(* IEC 61131-3 sources: verifaps-lib/iec-modularization/src/test/resources, 5 files *)

(* ---- program.st ---- *)
FUNCTION_BLOCK FB
VAR_INPUT
	x : INT;
END_VAR
VAR_OUTPUT
	y : INT;
END_VAR
	y := x+6;
END_FUNCTION_BLOCK

PROGRAM PGRM
VAR_INPUT
	x : INT;
END_VAR
VAR_OUTPUT
	y : INT;
END_VAR
VAR
	INST_FB : FB;
END_VAR
	INST_FB.x := 4;
	INST_FB();
	INST_FB.x := INST_FB.y + 2;
	INST_FB();
	y := INST_FB.y;
	IF x > 5 THEN
		y := 6;
	ELSEIF x > 3 THEN
		y := 7;
	ELSE
		y := x;
	END_IF
	y := y + 4;
END_PROGRAM

(* ---- program1.st ---- *)
TYPE
	TestEnum: (First, Second);
END_TYPE

FUNCTION_BLOCK BLOCK_A
	VAR_INPUT  x : INT; END_VAR
	VAR_OUTPUT y : INT; END_VAR
	y := x - INT#4;
END_FUNCTION_BLOCK

FUNCTION_BLOCK BLOCK_B
	VAR_INPUT  x : INT; END_VAR
	VAR_OUTPUT y : INT; END_VAR
	y := x + INT#6;
END_FUNCTION_BLOCK

FUNCTION_BLOCK TON
END_FUNCTION_BLOCK

PROGRAM PGRM
	VAR_INPUT  x      : INT;     END_VAR
	VAR_OUTPUT y      : INT;     END_VAR
	VAR        INST_A : BLOCK_A; END_VAR
	VAR        INST_B : BLOCK_B; END_VAR
	VAR        state  : TestEnum; END_VAR
	VAR  TestTimer : TON; END_VAR

	CASE state OF
		TestEnum#First:
			INST_A.x := INT#4;
		TestEnum#Second:
			INST_A.x := INT#8;
	END_CASE
	TestTimer();
	INST_A.x := x + INT#7;
	IF x > 5 THEN
		INST_A();
	END_IF

	INST_B.x := INST_A.y + INT#9;
	INST_B();

	y := INST_B.y;
END_PROGRAM

(* ---- program2.st ---- *)
FUNCTION_BLOCK BLOCK_A
	VAR_INPUT  x : INT; END_VAR
	VAR_OUTPUT y : INT; END_VAR
	y := x - INT#4;
END_FUNCTION_BLOCK

FUNCTION_BLOCK BLOCK_B
	VAR_INPUT  x : INT; END_VAR
	VAR_OUTPUT y : INT; END_VAR
	y := x + INT#3;
END_FUNCTION_BLOCK

PROGRAM PGRM
	VAR_INPUT  x      : INT;     END_VAR
	VAR_OUTPUT y      : INT;     END_VAR
	VAR        INST_A : BLOCK_A; END_VAR
	VAR        INST_B : BLOCK_B; END_VAR

	INST_A.x := x + INT#7;
	INST_A();

	INST_B.x := INST_A.y + INT#9;
	INST_B();

	y := INST_B.y + INT#3;
END_PROGRAM

(* ---- scenario0.st ---- *)
TYPE
    Magazin_states_t : (Green_Lamp , Init , Interstep , Magazin_Init , Magazin_Init_2 , Slider_Move_Back , Start_Magazin , Step0 , Step1 , convey);
    Crane_states_t : (Crane_Init , Crane_Init_2 , Crane_Lift_Conveyor , Crane_Lift_Magazine , Crane_On_Conveyor , Crane_Stop , Crane_Turn_Left , Init , Interstep , Interstep_2 , Interstep_Check_Workpiece , Magazin_Stop , Start_Crane , TimeDelay , Turn_Right , release);
END_TYPE

FUNCTION_BLOCK Magazin
    VAR_INPUT  CraneDown : BOOL; END_VAR
    VAR_INPUT  CraneOnConveyor : BOOL; END_VAR
    VAR_INPUT  CraneOnMagazin : BOOL; END_VAR
    VAR_INPUT  CraneSucked : BOOL; END_VAR
    VAR_INPUT  CraneUp : BOOL; END_VAR
    VAR_OUTPUT  MagazinGreenLamp : BOOL; END_VAR
    VAR_OUTPUT  MagazinSlider : BOOL; END_VAR
    VAR  SFCInit : BOOL; END_VAR
    VAR_INPUT  SFCReset : BOOL; END_VAR
    VAR_INPUT  SliderMovedOut : BOOL; END_VAR
    VAR_INPUT  SliderNotMovedOut : BOOL; END_VAR
    VAR_INPUT  StartButtonMagazin : BOOL; END_VAR
    VAR_OUTPUT  StartCommandMagazin : BOOL; END_VAR
    VAR_INPUT  StartVar : BOOL; END_VAR
    VAR_INPUT  WorkpieceReady : BOOL; END_VAR
    VAR  _state : Magazin_states_t; END_VAR
    VAR  _transit : BOOL; END_VAR
    VAR  interconnectMagazineStartCommand : BOOL; END_VAR

    CASE _state OF
        Magazin_states_t#Green_Lamp:
            _transit := FALSE;
            MagazinGreenLamp := TRUE;
            interconnectMagazineStartCommand := FALSE;
            IF TRUE THEN
                _transit := TRUE;
                _state := Magazin_states_t#Magazin_Init;
            END_IF;

        Magazin_states_t#Init:
            _transit := FALSE;
            IF TRUE THEN
                _transit := TRUE;
                _state := Magazin_states_t#Start_Magazin;
            END_IF;

        Magazin_states_t#Interstep:
            _transit := FALSE;
            StartCommandMagazin := TRUE;
            IF StartVar THEN
                _transit := TRUE;
                _state := Magazin_states_t#convey;
            END_IF;

        Magazin_states_t#Magazin_Init:
            _transit := FALSE;
            MagazinSlider := TRUE;
            IF TRUE THEN
                _transit := TRUE;
                _state := Magazin_states_t#Magazin_Init_2;
            END_IF;

        Magazin_states_t#Magazin_Init_2:
            _transit := FALSE;
            MagazinSlider := FALSE;
            IF TRUE THEN
                _transit := TRUE;
                _state := Magazin_states_t#Interstep;
            END_IF;

        Magazin_states_t#Slider_Move_Back:
            _transit := FALSE;
            IF ((SliderMovedOut = TRUE) AND (SliderNotMovedOut = FALSE)) THEN
                MagazinSlider := FALSE;
            END_IF;
            IF CraneUp THEN
                _transit := TRUE;
                _state := Magazin_states_t#Step1;
            END_IF;

        Magazin_states_t#Start_Magazin:
            _transit := FALSE;
            MagazinSlider := FALSE;
            MagazinGreenLamp := FALSE;
            StartVar := FALSE;
            StartCommandMagazin := FALSE;
            IF (StartButtonMagazin = TRUE) THEN
                interconnectMagazineStartCommand := TRUE;
            END_IF;
            IF interconnectMagazineStartCommand THEN
                _transit := TRUE;
                _state := Magazin_states_t#Green_Lamp;
            END_IF;

        Magazin_states_t#Step0:
            _transit := FALSE;
            IF CraneDown THEN
                _transit := TRUE;
                _state := Magazin_states_t#Slider_Move_Back;
            END_IF;

        Magazin_states_t#Step1:
            _transit := FALSE;
            IF CraneOnConveyor THEN
                _transit := TRUE;
                _state := Magazin_states_t#Interstep;
            END_IF;

        Magazin_states_t#convey:
            _transit := FALSE;
            IF SliderNotMovedOut THEN
                MagazinSlider := TRUE;
            END_IF;
            IF CraneOnMagazin THEN
                _transit := TRUE;
                _state := Magazin_states_t#Step0;
            END_IF;

            END_CASE
END_FUNCTION_BLOCK

FUNCTION_BLOCK Crane
    VAR_INPUT  CraneDown : BOOL; END_VAR
    VAR_OUTPUT  CraneLower : BOOL; END_VAR
    VAR_INPUT  CraneOnConveyor : BOOL; END_VAR
    VAR_INPUT  CraneOnMagazin : BOOL; END_VAR
    VAR_INPUT  CraneSucked : BOOL; END_VAR
    VAR_OUTPUT  CraneTurnClockwise : BOOL; END_VAR
    VAR_OUTPUT  CraneTurnCounterclockwise : BOOL; END_VAR
    VAR_INPUT  CraneUp : BOOL; END_VAR
    VAR_OUTPUT  MagazinVacuumOff : BOOL; END_VAR
    VAR_OUTPUT  MagazinVacuumOn : BOOL; END_VAR
    VAR  SFCInit : BOOL; END_VAR
    VAR_INPUT  SFCReset : BOOL; END_VAR
    VAR_INPUT  SliderMovedOut : BOOL; END_VAR
    VAR_INPUT  SliderNotMovedOut : BOOL; END_VAR
    VAR_INPUT  StartButtonMagazin : BOOL; END_VAR
    VAR_OUTPUT  StartCommandCrane : BOOL; END_VAR
    VAR_INPUT  StartVar : BOOL; END_VAR
    VAR  TimeDelay_Timer : TON; END_VAR
    VAR  TimeDelay_Timer_Duration : INT := INT#50; END_VAR
    VAR  TimeDelay_Timer_interconnect : BOOL; END_VAR
    VAR_INPUT  WorkpieceReady : BOOL; END_VAR
    VAR  _state : Crane_states_t; END_VAR
    VAR  _transit : BOOL; END_VAR
    VAR  interconnectCraneStartCommand : BOOL; END_VAR

    CASE _state OF
        Crane_states_t#Crane_Init:
            _transit := FALSE;
            CraneLower := TRUE;
            interconnectCraneStartCommand := FALSE;
            IF CraneDown THEN
                _transit := TRUE;
                _state := Crane_states_t#Crane_Init_2;
            END_IF;

        Crane_states_t#Crane_Init_2:
            _transit := FALSE;
            CraneLower := FALSE;
            IF CraneUp THEN
                _transit := TRUE;
                _state := Crane_states_t#Interstep;
            END_IF;

        Crane_states_t#Crane_Lift_Conveyor:
            _transit := FALSE;
            CraneLower := FALSE;
            IF TRUE THEN
                _transit := TRUE;
                _state := Crane_states_t#Interstep;
            END_IF;

        Crane_states_t#Crane_Lift_Magazine:
            _transit := FALSE;
            CraneLower := FALSE;
            IF CraneUp THEN
                _transit := TRUE;
                _state := Crane_states_t#Crane_Turn_Left;
            END_IF;

        Crane_states_t#Crane_On_Conveyor:
            _transit := FALSE;
            CraneTurnCounterclockwise := FALSE;
            CraneTurnClockwise := FALSE;
            CraneLower := TRUE;
            IF CraneDown THEN
                _transit := TRUE;
                _state := Crane_states_t#release;
            END_IF;

        Crane_states_t#Crane_Stop:
            _transit := FALSE;
            IF TRUE THEN
                _transit := TRUE;
                _state := Crane_states_t#Start_Crane;
            END_IF;

        Crane_states_t#Crane_Turn_Left:
            _transit := FALSE;
            CraneTurnCounterclockwise := TRUE;
            CraneTurnClockwise := FALSE;
            IF CraneOnConveyor THEN
                _transit := TRUE;
                _state := Crane_states_t#Crane_On_Conveyor;
            END_IF;

        Crane_states_t#Init:
            _transit := FALSE;
            IF TRUE THEN
                _transit := TRUE;
                _state := Crane_states_t#Start_Crane;
            END_IF;

        Crane_states_t#Interstep:
            _transit := FALSE;
            StartCommandCrane := TRUE;
            IF StartVar THEN
                _transit := TRUE;
                _state := Crane_states_t#Interstep_2;
            END_IF;

        Crane_states_t#Interstep_2:
            _transit := FALSE;
            IF SliderMovedOut THEN
                _transit := TRUE;
                _state := Crane_states_t#TimeDelay;
            END_IF;

        Crane_states_t#Interstep_Check_Workpiece:
            _transit := FALSE;
            IF WorkpieceReady THEN
                _transit := TRUE;
                _state := Crane_states_t#Magazin_Stop;
            ELSEIF NOT WorkpieceReady THEN
                _transit := TRUE;
                _state := Crane_states_t#Crane_Stop;
            END_IF;

        Crane_states_t#Magazin_Stop:
            _transit := FALSE;
            CraneTurnClockwise := FALSE;
            CraneTurnCounterclockwise := FALSE;
            MagazinVacuumOn := TRUE;
            MagazinVacuumOff := FALSE;
            CraneLower := TRUE;
            IF CraneSucked THEN
                _transit := TRUE;
                _state := Crane_states_t#Crane_Lift_Magazine;
            END_IF;

        Crane_states_t#Start_Crane:
            _transit := FALSE;
            CraneLower := FALSE;
            MagazinVacuumOff := TRUE;
            MagazinVacuumOn := FALSE;
            CraneTurnCounterclockwise := FALSE;
            CraneTurnClockwise := FALSE;
            StartVar := FALSE;
            StartCommandCrane := FALSE;
            IF (StartButtonMagazin = TRUE) THEN
                interconnectCraneStartCommand := TRUE;
            END_IF;
            IF interconnectCraneStartCommand THEN
                _transit := TRUE;
                _state := Crane_states_t#Crane_Init;
            END_IF;

        Crane_states_t#TimeDelay:
            _transit := FALSE;
            TimeDelay_Timer(IN := TRUE, PT := TimeDelay_Timer_Duration);
            TimeDelay_Timer_interconnect := TimeDelay_Timer.Q;
            IF TimeDelay_Timer_interconnect THEN
                _transit := TRUE;
                _state := Crane_states_t#Turn_Right;
            END_IF;

        Crane_states_t#Turn_Right:
            _transit := FALSE;
            CraneTurnClockwise := TRUE;
            CraneTurnCounterclockwise := FALSE;
            IF CraneOnMagazin THEN
                _transit := TRUE;
                _state := Crane_states_t#Interstep_Check_Workpiece;
            END_IF;

        Crane_states_t#release:
            _transit := FALSE;
            MagazinVacuumOff := TRUE;
            MagazinVacuumOn := FALSE;
            IF TRUE THEN
                _transit := TRUE;
                _state := Crane_states_t#Crane_Lift_Conveyor;
            END_IF;

            END_CASE
END_FUNCTION_BLOCK

PROGRAM Main

VAR_OUTPUT  Actuator_CraneLower : BOOL; END_VAR
VAR_OUTPUT  Actuator_CraneTurnClockwise : BOOL; END_VAR
VAR_OUTPUT  Actuator_CraneTurnCounterclockwise : BOOL; END_VAR
VAR_OUTPUT  Actuator_MagazinGreenLamp : BOOL; END_VAR
VAR_OUTPUT  Actuator_MagazinSlider : BOOL; END_VAR
VAR_OUTPUT  Actuator_MagazinVacuumOff : BOOL; END_VAR
VAR_OUTPUT  Actuator_MagazinVacuumOn : BOOL; END_VAR
VAR_OUTPUT  Actuator_MagazinWhiteLamp : BOOL; END_VAR
VAR  Crane : Crane; END_VAR
VAR  Mag : Magazin; END_VAR
VAR_INPUT  Sensor_CraneDown : BOOL; END_VAR
VAR_INPUT  Sensor_CraneOnConveyor : BOOL; END_VAR
VAR_INPUT  Sensor_CraneOnMagazin : BOOL; END_VAR
VAR_INPUT  Sensor_CranePosition : BOOL; END_VAR
VAR_INPUT  Sensor_CraneSucked : BOOL; END_VAR
VAR_INPUT  Sensor_CraneUp : BOOL; END_VAR
VAR_INPUT  Sensor_MagazinEmergencyStop : BOOL; END_VAR
VAR_INPUT  Sensor_MagazinSwitchManuellAutomatic : BOOL; END_VAR
VAR_INPUT  Sensor_SliderMovedOut : BOOL; END_VAR
VAR_INPUT  Sensor_SliderNotMovedOut : BOOL; END_VAR
VAR_INPUT  Sensor_StartButtonMagazin : BOOL; END_VAR
VAR_INPUT  Sensor_WorkpieceReady : BOOL; END_VAR
Mag.SliderNotMovedOut := Sensor_SliderNotMovedOut;
Mag.SliderMovedOut := Sensor_SliderMovedOut;
Mag.CraneOnMagazin := Sensor_CraneOnMagazin;
Mag.CraneDown := Sensor_CraneDown;
Mag.CraneUp := Sensor_CraneUp;
Mag.CraneOnConveyor := Sensor_CraneOnConveyor;
Mag.WorkpieceReady := Sensor_WorkpieceReady;
Mag.StartButtonMagazin := Sensor_StartButtonMagazin;
Actuator_MagazinSlider := Mag.MagazinSlider;
Actuator_MagazinGreenLamp := Mag.MagazinGreenLamp;
Crane.WorkpieceReady := Sensor_WorkpieceReady;
Crane.CraneUp := Sensor_CraneUp;
Crane.CraneOnConveyor := Sensor_CraneOnConveyor;
Crane.CraneDown := Sensor_CraneDown;
Crane.CraneSucked := Sensor_CraneSucked;
Crane.CraneOnMagazin := Sensor_CraneOnMagazin;
Crane.SliderMovedOut := Sensor_SliderMovedOut;
Crane.StartButtonMagazin := Sensor_StartButtonMagazin;
Actuator_CraneTurnCounterclockwise := Crane.CraneTurnCounterclockwise;
Actuator_CraneTurnClockwise := Crane.CraneTurnClockwise;
Actuator_CraneLower := Crane.CraneLower;
Actuator_MagazinVacuumOff := Crane.MagazinVacuumOff;
Actuator_MagazinVacuumOn := Crane.MagazinVacuumOn;
IF Sensor_MagazinEmergencyStop THEN
    Mag();
    Crane();
    IF Actuator_MagazinGreenLamp THEN
        IF (Crane.StartCommandCrane AND Mag.StartCommandMagazin) THEN
            Crane.StartVar := TRUE;
            Mag.StartVar := TRUE;
        END_IF;
    END_IF;
    Crane.SFCReset := FALSE;
    Mag.SFCReset := FALSE;
ELSEIF NOT Sensor_MagazinEmergencyStop THEN
    Actuator_MagazinSlider := FALSE;
    Actuator_CraneLower := FALSE;
    Actuator_MagazinVacuumOn := FALSE;
    Actuator_MagazinVacuumOff := TRUE;
    Actuator_MagazinGreenLamp := FALSE;
    Actuator_CraneTurnCounterclockwise := FALSE;
    Actuator_CraneTurnClockwise := FALSE;
    Crane.SFCReset := TRUE;
    Mag.SFCReset := TRUE;
    Crane.StartVar := FALSE;
    Mag.StartVar := FALSE;
END_IF
END_PROGRAM

FUNCTION_BLOCK TON

VAR_INPUT
    IN : BOOL;
    PT : USINT;
END_VAR

VAR_OUTPUT
    Q  : BOOL;
    ET : USINT;
END_VAR

IF IN THEN
    Q:= ET = USINT#0;
    IF ET > USINT#0 THEN
        ET := ET - USINT#1;
    ELSE
        ET := USINT#0;
    END_IF
ELSE
    Q  := FALSE;
    ET := PT;
END_IF

END_FUNCTION_BLOCK

(* ---- scenario1.st ---- *)
TYPE
    Magazin_states_t : (Green_Lamp , Init , Interstep , Magazin_Init , Magazin_Init_2 , Slider_Move_Back , Start_Magazin , Step0 , Step1 , convey);
    Crane_states_t : (Crane_Init , Crane_Init_2 , Crane_Lift_Conveyor , Crane_Lift_Magazine , Crane_On_Conveyor , Crane_Stop , Crane_Turn_Left , Init , Interstep , Interstep_2 , Interstep_Check_Workpiece , Magazin_Stop , Start_Crane , TimeDelay , Turn_Right , release);
END_TYPE

FUNCTION_BLOCK Magazin
    VAR_INPUT  CraneDown : BOOL; END_VAR
    VAR_INPUT  CraneOnConveyor : BOOL; END_VAR
    VAR_INPUT  CraneOnMagazin : BOOL; END_VAR
    VAR_INPUT  CraneSucked : BOOL; END_VAR
    VAR_INPUT  CraneUp : BOOL; END_VAR
    VAR_OUTPUT  MagazinGreenLamp : BOOL; END_VAR
    VAR_OUTPUT  MagazinSlider : BOOL; END_VAR
    VAR  SFCInit : BOOL; END_VAR
    VAR_INPUT  SFCReset : BOOL; END_VAR
    VAR_INPUT  SliderMovedOut : BOOL; END_VAR
    VAR_INPUT  SliderNotMovedOut : BOOL; END_VAR
    VAR_INPUT  StartButtonMagazin : BOOL; END_VAR
    VAR_OUTPUT  StartCommandMagazin : BOOL; END_VAR
    VAR_INPUT  StartVar : BOOL; END_VAR
    VAR_INPUT  WorkpieceReady : BOOL; END_VAR
    VAR  _state : Magazin_states_t; END_VAR
    VAR  _transit : BOOL; END_VAR
    VAR  interconnectMagazinStartCommand : BOOL; END_VAR

    CASE _state OF
        Magazin_states_t#Green_Lamp:
            _transit := FALSE;
            MagazinGreenLamp := TRUE;
            interconnectMagazinStartCommand := FALSE;
            IF TRUE THEN
                _transit := TRUE;
                _state := Magazin_states_t#Magazin_Init;
            END_IF;

        Magazin_states_t#Init:
            _transit := FALSE;
            IF TRUE THEN
                _transit := TRUE;
                _state := Magazin_states_t#Start_Magazin;
            END_IF;

        Magazin_states_t#Interstep:
            _transit := FALSE;
            StartCommandMagazin := TRUE;
            IF StartVar THEN
                _transit := TRUE;
                _state := Magazin_states_t#convey;
            END_IF;

        Magazin_states_t#Magazin_Init:
            _transit := FALSE;
            MagazinSlider := TRUE;
            IF TRUE THEN
                _transit := TRUE;
                _state := Magazin_states_t#Magazin_Init_2;
            END_IF;

        Magazin_states_t#Magazin_Init_2:
            _transit := FALSE;
            MagazinSlider := FALSE;
            IF TRUE THEN
                _transit := TRUE;
                _state := Magazin_states_t#Interstep;
            END_IF;

        Magazin_states_t#Slider_Move_Back:
            _transit := FALSE;
            IF ((SliderMovedOut = TRUE) AND (SliderNotMovedOut = FALSE)) THEN
                MagazinSlider := FALSE;
            END_IF;
            IF CraneUp THEN
                _transit := TRUE;
                _state := Magazin_states_t#Step1;
            END_IF;

        Magazin_states_t#Start_Magazin:
            _transit := FALSE;
            MagazinSlider := FALSE;
            MagazinGreenLamp := FALSE;
            StartVar := FALSE;
            StartCommandMagazin := FALSE;
            IF (StartButtonMagazin = TRUE) THEN
                interconnectMagazinStartCommand := TRUE;
            END_IF;
            IF interconnectMagazinStartCommand THEN
                _transit := TRUE;
                _state := Magazin_states_t#Green_Lamp;
            END_IF;

        Magazin_states_t#Step0:
            _transit := FALSE;
            IF CraneDown THEN
                _transit := TRUE;
                _state := Magazin_states_t#Slider_Move_Back;
            END_IF;

        Magazin_states_t#Step1:
            _transit := FALSE;
            IF CraneOnConveyor THEN
                _transit := TRUE;
                _state := Magazin_states_t#Interstep;
            END_IF;

        Magazin_states_t#convey:
            _transit := FALSE;
            IF SliderNotMovedOut THEN
                MagazinSlider := TRUE;
            END_IF;
            IF CraneOnMagazin THEN
                _transit := TRUE;
                _state := Magazin_states_t#Step0;
            END_IF;

            END_CASE
END_FUNCTION_BLOCK

PROGRAM Main

VAR_OUTPUT  Actuator_CraneLower : BOOL; END_VAR
VAR_OUTPUT  Actuator_CraneTurnClockwise : BOOL; END_VAR
VAR_OUTPUT  Actuator_CraneTurnCounterclockwise : BOOL; END_VAR
VAR_OUTPUT  Actuator_MagazinGreenLamp : BOOL; END_VAR
VAR_OUTPUT  Actuator_MagazinSlider : BOOL; END_VAR
VAR_OUTPUT  Actuator_MagazinVacuumOff : BOOL; END_VAR
VAR_OUTPUT  Actuator_MagazinVacuumOn : BOOL; END_VAR
VAR_OUTPUT  Actuator_MagazinWhiteLamp : BOOL; END_VAR
VAR  Crane : Crane; END_VAR
VAR  Mag : Magazin; END_VAR
VAR_INPUT  Sensor_CraneDown : BOOL; END_VAR
VAR_INPUT  Sensor_CraneOnConveyor : BOOL; END_VAR
VAR_INPUT  Sensor_CraneOnMagazin : BOOL; END_VAR
VAR_INPUT  Sensor_CranePosition : BOOL; END_VAR
VAR_INPUT  Sensor_CraneSucked : BOOL; END_VAR
VAR_INPUT  Sensor_CraneUp : BOOL; END_VAR
VAR_INPUT  Sensor_MagazinEmergencyStop : BOOL; END_VAR
VAR_INPUT  Sensor_MagazinSwitchManuellAutomatic : BOOL; END_VAR
VAR_INPUT  Sensor_SliderMovedOut : BOOL; END_VAR
VAR_INPUT  Sensor_SliderNotMovedOut : BOOL; END_VAR
VAR_INPUT  Sensor_StartButtonMagazin : BOOL; END_VAR
VAR_INPUT  Sensor_WorkpieceReady : BOOL; END_VAR
Mag.SliderNotMovedOut := Sensor_SliderNotMovedOut;
Mag.SliderMovedOut := Sensor_SliderMovedOut;
Mag.CraneOnMagazin := Sensor_CraneOnMagazin;
Mag.CraneDown := Sensor_CraneDown;
Mag.CraneUp := Sensor_CraneUp;
Mag.CraneOnConveyor := Sensor_CraneOnConveyor;
Mag.WorkpieceReady := Sensor_WorkpieceReady;
Mag.StartButtonMagazin := Sensor_StartButtonMagazin;
Actuator_MagazinSlider := Mag.MagazinSlider;
Actuator_MagazinGreenLamp := Mag.MagazinGreenLamp;
Crane.WorkpieceReady := Sensor_WorkpieceReady;
Crane.CraneUp := Sensor_CraneUp;
Crane.CraneOnConveyor := Sensor_CraneOnConveyor;
Crane.CraneDown := Sensor_CraneDown;
Crane.CraneSucked := Sensor_CraneSucked;
Crane.CraneOnMagazin := Sensor_CraneOnMagazin;
Crane.SliderMovedOut := Sensor_SliderMovedOut;
Crane.StartButtonMagazin := Sensor_StartButtonMagazin;
Actuator_CraneTurnCounterclockwise := Crane.CraneTurnCounterclockwise;
Actuator_CraneTurnClockwise := Crane.CraneTurnClockwise;
Actuator_CraneLower := Crane.CraneLower;
Actuator_MagazinVacuumOff := Crane.MagazinVacuumOff;
Actuator_MagazinVacuumOn := Crane.MagazinVacuumOn;
IF Sensor_MagazinEmergencyStop THEN
    Mag();
    Crane();
    IF Actuator_MagazinGreenLamp THEN
        IF (Crane.StartCommandCrane AND Mag.StartCommandMagazin) THEN
            Crane.StartVar := TRUE;
            Mag.StartVar := TRUE;
        END_IF;
    END_IF;
    Crane.SFCReset := FALSE;
    Mag.SFCReset := FALSE;
ELSEIF NOT Sensor_MagazinEmergencyStop THEN
    Actuator_MagazinSlider := FALSE;
    Actuator_CraneLower := FALSE;
    Actuator_MagazinVacuumOn := FALSE;
    Actuator_MagazinVacuumOff := TRUE;
    Actuator_MagazinGreenLamp := FALSE;
    Actuator_CraneTurnCounterclockwise := FALSE;
    Actuator_CraneTurnClockwise := FALSE;
    Crane.SFCReset := TRUE;
    Mag.SFCReset := TRUE;
    Crane.StartVar := FALSE;
    Mag.StartVar := FALSE;
END_IF
END_PROGRAM
FUNCTION_BLOCK Crane
VAR_INPUT  CraneDown : BOOL; END_VAR
VAR_OUTPUT  CraneLower : BOOL; END_VAR
VAR_INPUT  CraneOnConveyor : BOOL; END_VAR
VAR_INPUT  CraneOnMagazin : BOOL; END_VAR
VAR_INPUT  CraneSucked : BOOL; END_VAR
VAR_OUTPUT  CraneTurnClockwise : BOOL; END_VAR
VAR_OUTPUT  CraneTurnCounterclockwise : BOOL; END_VAR
VAR_INPUT  CraneUp : BOOL; END_VAR
VAR_OUTPUT  MagazinVacuumOff : BOOL; END_VAR
VAR_OUTPUT  MagazinVacuumOn : BOOL; END_VAR
VAR  SFCInit : BOOL; END_VAR
VAR_INPUT  SFCReset : BOOL; END_VAR
VAR_INPUT  SliderMovedOut : BOOL; END_VAR
VAR_INPUT  SliderNotMovedOut : BOOL; END_VAR
VAR_INPUT  StartButtonMagazin : BOOL; END_VAR
VAR_OUTPUT  StartCommandCrane : BOOL; END_VAR
VAR_INPUT  StartVar : BOOL; END_VAR
VAR  TimeDelay_Timer : TON; END_VAR
VAR  TimeDelay_Timer_Duration : INT := INT#50; END_VAR
VAR  TimeDelay_Timer_interconnect : BOOL; END_VAR
VAR_INPUT  WorkpieceReady : BOOL; END_VAR
VAR  _state : Crane_states_t; END_VAR
VAR  _transit : BOOL; END_VAR
VAR  interconnectCraneStartCommand : BOOL; END_VAR

CASE _state OF
    Crane_states_t#Crane_Init:
        _transit := FALSE;
        CraneLower := TRUE;
        interconnectCraneStartCommand := FALSE;
        IF CraneDown THEN
            _transit := TRUE;
            _state := Crane_states_t#Crane_Init_2;
        END_IF;

    Crane_states_t#Crane_Init_2:
        _transit := FALSE;
        CraneLower := FALSE;
        IF CraneUp THEN
            _transit := TRUE;
            _state := Crane_states_t#Interstep;
        END_IF;

    Crane_states_t#Crane_Lift_Conveyor:
        _transit := FALSE;
        CraneLower := FALSE;
        IF TRUE THEN
            _transit := TRUE;
            _state := Crane_states_t#Interstep;
        END_IF;

    Crane_states_t#Crane_Lift_Magazine:
        _transit := FALSE;
        CraneLower := FALSE;
        IF CraneUp THEN
            _transit := TRUE;
            _state := Crane_states_t#Crane_Turn_Left;
        END_IF;

    Crane_states_t#Crane_On_Conveyor:
        _transit := FALSE;
        CraneTurnCounterclockwise := FALSE;
        CraneTurnClockwise := FALSE;
        CraneLower := TRUE;
        IF CraneDown THEN
            _transit := TRUE;
            _state := Crane_states_t#release;
        END_IF;

    Crane_states_t#Crane_Stop:
        _transit := FALSE;
        IF TRUE THEN
            _transit := TRUE;
            _state := Crane_states_t#Start_Crane;
        END_IF;

    Crane_states_t#Crane_Turn_Left:
        _transit := FALSE;
        CraneTurnCounterclockwise := TRUE;
        CraneTurnClockwise := FALSE;
        IF CraneOnConveyor THEN
            _transit := TRUE;
            _state := Crane_states_t#Crane_On_Conveyor;
        END_IF;

    Crane_states_t#Init:
        _transit := FALSE;
        IF TRUE THEN
            _transit := TRUE;
            _state := Crane_states_t#Start_Crane;
        END_IF;

    Crane_states_t#Interstep:
        _transit := FALSE;
        StartCommandCrane := TRUE;
        IF StartVar THEN
            _transit := TRUE;
            _state := Crane_states_t#Interstep_2;
        END_IF;

    Crane_states_t#Interstep_2:
        _transit := FALSE;
        IF SliderMovedOut THEN
            _transit := TRUE;
            _state := Crane_states_t#TimeDelay;
        END_IF;

    Crane_states_t#Interstep_Check_Workpiece:
        _transit := FALSE;
        IF WorkpieceReady THEN
            _transit := TRUE;
            _state := Crane_states_t#Magazin_Stop;
        ELSEIF NOT WorkpieceReady THEN
            _transit := TRUE;
            _state := Crane_states_t#Crane_Stop;
        END_IF;

    Crane_states_t#Magazin_Stop:
        _transit := FALSE;
        CraneTurnClockwise := FALSE;
        CraneTurnCounterclockwise := FALSE;
        MagazinVacuumOn := TRUE;
        MagazinVacuumOff := FALSE;
        CraneLower := TRUE;
        IF CraneSucked THEN
            _transit := TRUE;
            _state := Crane_states_t#Crane_Lift_Magazine;
        END_IF;

    Crane_states_t#Start_Crane:
        _transit := FALSE;
        CraneLower := FALSE;
        MagazinVacuumOff := TRUE;
        MagazinVacuumOn := FALSE;
        CraneTurnCounterclockwise := FALSE;
        CraneTurnClockwise := FALSE;
        StartVar := FALSE;
        StartCommandCrane := FALSE;
        IF (StartButtonMagazin = TRUE) THEN
            interconnectCraneStartCommand := TRUE;
        END_IF;
        IF interconnectCraneStartCommand THEN
            _transit := TRUE;
            _state := Crane_states_t#Crane_Init;
        END_IF;

    Crane_states_t#TimeDelay:
        _transit := FALSE;
        TimeDelay_Timer(IN := TRUE, PT := TimeDelay_Timer_Duration);
        TimeDelay_Timer_interconnect := TimeDelay_Timer.Q;
        IF TimeDelay_Timer_interconnect THEN
            _transit := TRUE;
            _state := Crane_states_t#Turn_Right;
        END_IF;

    Crane_states_t#Turn_Right:
        _transit := FALSE;
        CraneTurnClockwise := TRUE;
        CraneTurnCounterclockwise := FALSE;
        IF CraneOnMagazin THEN
            _transit := TRUE;
            _state := Crane_states_t#Interstep_Check_Workpiece;
        END_IF;

    Crane_states_t#release:
        _transit := FALSE;
        MagazinVacuumOff := TRUE;
        MagazinVacuumOn := FALSE;
        IF TRUE THEN
            _transit := TRUE;
            _state := Crane_states_t#Crane_Lift_Conveyor;
        END_IF;

    END_CASE
END_FUNCTION_BLOCK

FUNCTION_BLOCK TON

VAR_INPUT
    IN : BOOL;
    PT : USINT;
END_VAR

VAR_OUTPUT
    Q  : BOOL;
    ET : USINT;
END_VAR

IF IN THEN
    Q:= ET = USINT#0;
    IF ET > USINT#0 THEN
        ET := ET - USINT#1;
    ELSE
        ET := USINT#0;
    END_IF
ELSE
    Q  := FALSE;
    ET := PT;
END_IF

END_FUNCTION_BLOCK
